{attribute 'GeneratedUsingTerminal: EP1859-0042-0018'}
{attribute addProperty BoxType "EP1859-0042-0018"}
{attribute addProperty Id "OutputAT %Q*BOOL1"}
{attribute addProperty CRC "1120571895"}
{attribute addProperty Size "1"}
TYPE DO_X08_Pin_42CA91F7 EXTENDS OutputBase_10CEE7DE :
STRUCT
	{attribute addProperty Name "Output"}
	Output AT %Q* : BOOL;
END_STRUCT
END_TYPE

(* stored: Version 1.2.0.0, ProductVersion 3.1.4024.11
   DUT DO_X08_Pin_42CA91F7: Id {13a17057-3a66-4a3f-93ef-96cd5b1b112b} *)
